// TIA Portal V17 export
BLOCK "Main"   // ObjectSW1, LAD
// Cyclic main OB
BEGIN

REGION Network 1: Run motor control
END_REGION
END_BLOCK
